INTERFACE I_AxisMoveVelocity EXTENDS I_Base

METHOD MoveVelocity : BOOL
VAR_INPUT
	Velocity	  : LREAL;
	AbortPrevious : BOOL := TRUE;
END_VAR
END_METHOD

END_INTERFACE

(* stored: Version 1.1.0.1, ProductVersion 3.1.4026.18
   Itf I_AxisMoveVelocity: Id {8cee7583-ea15-463b-88b6-009ca18897f0}
   Method MoveVelocity: Id {73d31342-a8a2-4aa7-9f5d-170d9fb4ee21} *)
